FUNCTION_BLOCK FB_TemplateSimpleDevice EXTENDS FB_Base
VAR_INPUT
END_VAR
VAR_OUTPUT
END_VAR
VAR
END_VAR

//FB_Init ist immer implizit verfügbar und wird primär für die Initialisierung verwendet.
//Der Rückgabewert wird nicht ausgewertet. Für gezielte Einflussnahme können Sie
//die Methoden explizit deklarieren und darin mit dem Standard-Initialisierungscode 
//zusätzlichen Code bereitstellen. Sie können den Rückgabewert auswerten.
METHOD FB_Init: BOOL
VAR_INPUT    
	bInitRetains					: BOOL; 					// TRUE: Die Retain-Variablen werden initialisiert (Reset warm / Reset kalt)    
	bInCopyCode						: BOOL;  					// TRUE: Die Instanz wird danach in den Kopiercode kopiert (Online-Change)
	
	I_Name                : STRING;         //  Name
	I_ID                  : UINT;            // ID
END_VAR
END_METHOD

END_FUNCTION_BLOCK

(* stored: Version 1.1.0.1, ProductVersion 3.1.4026.18
   POU FB_TemplateSimpleDevice: Id {42f4f954-a23c-4534-a4a1-5c581f1295d3}, SpecialFunc None
   Folder 01 Properties: Id {fdf4616f-ac96-41a0-9463-60f0af68be40}
   Folder 02 Methodes: Id {c79d2a39-5faa-4f3e-bd34-705513f2dce8}
   Method FB_Init: Id {d6e295d7-025a-456c-9ea7-de11ad1dfba8} *)
